    movel([0.147581, -1.249692, -2.655126, -0.807572, 1.570796, 1.718377],accel_mss,speed_ms,0,blend_radius_m)
    movel([0.147363, -1.250802, -2.654535, -0.807052, 1.570796, 1.718159],accel_mss,speed_ms,0,blend_radius_m)
    movel([0.147089, -1.251643, -2.654086, -0.806660, 1.570796, 1.717886],accel_mss,speed_ms,0,blend_radius_m)
    movel([0.145883, -1.253778, -2.652943, -0.805668, 1.570796, 1.716679],accel_mss,speed_ms,0,blend_radius_m)
    movel([0.144114, -1.255772, -2.651871, -0.804746, 1.570796, 1.714911],accel_mss,speed_ms,0,blend_radius_m)
    movel([0.142022, -1.257371, -2.651008, -0.804011, 1.570796, 1.712819],accel_mss,speed_ms,0,blend_radius_m)
    movel([0.139874, -1.258370, -2.650466, -0.803552, 1.570796, 1.710670],accel_mss,speed_ms,0,blend_radius_m)
    movel([0.139347, -1.258581, -2.650352, -0.803456, 1.570796, 1.710143],accel_mss,speed_ms,0,blend_radius_m)
    movel([0.139026, -1.258793, -2.650237, -0.803359, 1.570796, 1.709822],accel_mss,speed_ms,0,blend_radius_m)
    movel([0.138790, -1.259384, -2.649916, -0.803089, 1.570796, 1.709586],accel_mss,speed_ms,0,blend_radius_m)
    movel([0.138626, -1.259915, -2.649627, -0.802847, 1.570796, 1.709423],accel_mss,speed_ms,0,blend_radius_m)
    movel([0.138465, -1.260505, -2.649306, -0.802578, 1.570796, 1.709261],accel_mss,speed_ms,0,blend_radius_m)
    movel([0.138304, -1.261095, -2.648985, -0.802310, 1.570796, 1.709100],accel_mss,speed_ms,0,blend_radius_m)
    movel([0.138138, -1.261625, -2.648695, -0.802069, 1.570796, 1.708934],accel_mss,speed_ms,0,blend_radius_m)
    movel([0.137986, -1.262068, -2.648453, -0.801868, 1.570796, 1.708782],accel_mss,speed_ms,0,blend_radius_m)
    movel([0.137718, -1.262390, -2.648277, -0.801722, 1.570796, 1.708514],accel_mss,speed_ms,0,blend_radius_m)
    movel([0.137358, -1.262485, -2.648225, -0.801679, 1.570796, 1.708154],accel_mss,speed_ms,0,blend_radius_m)
    speed_ms = 0.003
    movel([0.137358, -1.248347, -2.641414, -0.822628, 1.570796, 1.708154],accel_mss,speed_ms,0,blend_radius_m)
    speed_ms = 1.000
    movel([0.137358, -1.221519, -2.627413, -0.863457, 1.570796, 1.708154],accel_mss,speed_ms,0,blend_radius_m)
    movel([0.136331, -1.221369, -2.627491, -0.863529, 1.570796, 1.707127],accel_mss,speed_ms,0,blend_radius_m)
    movel([0.136331, -1.248198, -2.641494, -0.822697, 1.570796, 1.707127],accel_mss,speed_ms,0,blend_radius_m)
    speed_ms = 0.003
    movel([0.136331, -1.258756, -2.646615, -0.807017, 1.570796, 1.707127],accel_mss,speed_ms,0,blend_radius_m)
    speed_ms = 0.007
    movel([0.135965, -1.259022, -2.646471, -0.806896, 1.570796, 1.706761],accel_mss,speed_ms,0,blend_radius_m)
    movel([0.135639, -1.258950, -2.646510, -0.806929, 1.570796, 1.706435],accel_mss,speed_ms,0,blend_radius_m)
    movel([0.135615, -1.258574, -2.646715, -0.807101, 1.570796, 1.706412],accel_mss,speed_ms,0,blend_radius_m)
    movel([0.136097, -1.255221, -2.648532, -0.808636, 1.570796, 1.706894],accel_mss,speed_ms,0,blend_radius_m)
    movel([0.136603, -1.251789, -2.650378, -0.810222, 1.570796, 1.707400],accel_mss,speed_ms,0,blend_radius_m)
    movel([0.136724, -1.251497, -2.650534, -0.810358, 1.570796, 1.707521],accel_mss,speed_ms,0,blend_radius_m)
    movel([0.137247, -1.251196, -2.650695, -0.810498, 1.570796, 1.708044],accel_mss,speed_ms,0,blend_radius_m)
    movel([0.137587, -1.251126, -2.650733, -0.810530, 1.570796, 1.708383],accel_mss,speed_ms,0,blend_radius_m)
    movel([0.137884, -1.251389, -2.650592, -0.810408, 1.570796, 1.708680],accel_mss,speed_ms,0,blend_radius_m)
    movel([0.137821, -1.251968, -2.650282, -0.810139, 1.570796, 1.708618],accel_mss,speed_ms,0,blend_radius_m)
    movel([0.137622, -1.253027, -2.649713, -0.809648, 1.570796, 1.708419],accel_mss,speed_ms,0,blend_radius_m)
    movel([0.137096, -1.255476, -2.648394, -0.808519, 1.570796, 1.707892],accel_mss,speed_ms,0,blend_radius_m)
    movel([0.136830, -1.256677, -2.647744, -0.807968, 1.570796, 1.707626],accel_mss,speed_ms,0,blend_radius_m)
    movel([0.136591, -1.257717, -2.647180, -0.807492, 1.570796, 1.707388],accel_mss,speed_ms,0,blend_radius_m)
    movel([0.136382, -1.258618, -2.646691, -0.807081, 1.570796, 1.707178],accel_mss,speed_ms,0,blend_radius_m)
    speed_ms = 0.003
    movel([0.136331, -1.262337, -2.648306, -0.801746, 1.570796, 1.707127],accel_mss,speed_ms,0,blend_radius_m)
    speed_ms = 0.007
    movel([0.135965, -1.262602, -2.648161, -0.801626, 1.570796, 1.706761],accel_mss,speed_ms,0,blend_radius_m)
    movel([0.135639, -1.262530, -2.648201, -0.801659, 1.570796, 1.706435],accel_mss,speed_ms,0,blend_radius_m)
    movel([0.135615, -1.262155, -2.648406, -0.801828, 1.570796, 1.706412],accel_mss,speed_ms,0,blend_radius_m)
    movel([0.136097, -1.258809, -2.650228, -0.803352, 1.570796, 1.706894],accel_mss,speed_ms,0,blend_radius_m)
    movel([0.136603, -1.255383, -2.652081, -0.804926, 1.570796, 1.707400],accel_mss,speed_ms,0,blend_radius_m)
    movel([0.136724, -1.255092, -2.652237, -0.805060, 1.570796, 1.707521],accel_mss,speed_ms,0,blend_radius_m)
    movel([0.137247, -1.254791, -2.652399, -0.805199, 1.570796, 1.708044],accel_mss,speed_ms,0,blend_radius_m)
    movel([0.137587, -1.254721, -2.652437, -0.805231, 1.570796, 1.708383],accel_mss,speed_ms,0,blend_radius_m)
    movel([0.137884, -1.254983, -2.652296, -0.805110, 1.570796, 1.708680],accel_mss,speed_ms,0,blend_radius_m)
    movel([0.137821, -1.255562, -2.651984, -0.804843, 1.570796, 1.708618],accel_mss,speed_ms,0,blend_radius_m)
    movel([0.137622, -1.256619, -2.651414, -0.804356, 1.570796, 1.708419],accel_mss,speed_ms,0,blend_radius_m)
    movel([0.137096, -1.259063, -2.650090, -0.803235, 1.570796, 1.707892],accel_mss,speed_ms,0,blend_radius_m)
    movel([0.136830, -1.260262, -2.649439, -0.802689, 1.570796, 1.707626],accel_mss,speed_ms,0,blend_radius_m)
    movel([0.136591, -1.261299, -2.648873, -0.802217, 1.570796, 1.707388],accel_mss,speed_ms,0,blend_radius_m)
    movel([0.136382, -1.262199, -2.648382, -0.801809, 1.570796, 1.707178],accel_mss,speed_ms,0,blend_radius_m)
    speed_ms = 0.003
    movel([0.136331, -1.248198, -2.641494, -0.822697, 1.570796, 1.707127],accel_mss,speed_ms,0,blend_radius_m)
    speed_ms = 1.000
    movel([0.136331, -1.221369, -2.627491, -0.863529, 1.570796, 1.707127],accel_mss,speed_ms,0,blend_radius_m)
    movel([0.135518, -1.213284, -2.631635, -0.867470, 1.570796, 1.706315],accel_mss,speed_ms,0,blend_radius_m)
    movel([0.135518, -1.240201, -2.645745, -0.826443, 1.570796, 1.706315],accel_mss,speed_ms,0,blend_radius_m)
    speed_ms = 0.003
    movel([0.135518, -1.250801, -2.650907, -0.810681, 1.570796, 1.706315],accel_mss,speed_ms,0,blend_radius_m)
    speed_ms = 0.007
    movel([0.135184, -1.250928, -2.650838, -0.810622, 1.570796, 1.705981],accel_mss,speed_ms,0,blend_radius_m)
    movel([0.134896, -1.250953, -2.650826, -0.810611, 1.570796, 1.705692],accel_mss,speed_ms,0,blend_radius_m)
    movel([0.134573, -1.250950, -2.650827, -0.810612, 1.570796, 1.705369],accel_mss,speed_ms,0,blend_radius_m)
    movel([0.134262, -1.250915, -2.650845, -0.810628, 1.570796, 1.705059],accel_mss,speed_ms,0,blend_radius_m)
    movel([0.133875, -1.250842, -2.650884, -0.810662, 1.570796, 1.704671],accel_mss,speed_ms,0,blend_radius_m)
    movel([0.133663, -1.250756, -2.650931, -0.810702, 1.570796, 1.704460],accel_mss,speed_ms,0,blend_radius_m)
    movel([0.133527, -1.250440, -2.651099, -0.810849, 1.570796, 1.704323],accel_mss,speed_ms,0,blend_radius_m)
    movel([0.133693, -1.249935, -2.651369, -0.811085, 1.570796, 1.704489],accel_mss,speed_ms,0,blend_radius_m)
    movel([0.134107, -1.249492, -2.651605, -0.811291, 1.570796, 1.704903],accel_mss,speed_ms,0,blend_radius_m)
    movel([0.134658, -1.249246, -2.651736, -0.811407, 1.570796, 1.705455],accel_mss,speed_ms,0,blend_radius_m)
    movel([0.135181, -1.249271, -2.651723, -0.811395, 1.570796, 1.705978],accel_mss,speed_ms,0,blend_radius_m)
    movel([0.135427, -1.249443, -2.651631, -0.811314, 1.570796, 1.706223],accel_mss,speed_ms,0,blend_radius_m)
    movel([0.135661, -1.249807, -2.651437, -0.811145, 1.570796, 1.706457],accel_mss,speed_ms,0,blend_radius_m)
    movel([0.135822, -1.250215, -2.651220, -0.810954, 1.570796, 1.706618],accel_mss,speed_ms,0,blend_radius_m)
    movel([0.135808, -1.250511, -2.651062, -0.810817, 1.570796, 1.706604],accel_mss,speed_ms,0,blend_radius_m)
    movel([0.135518, -1.250801, -2.650907, -0.810681, 1.570796, 1.706315],accel_mss,speed_ms,0,blend_radius_m)
    speed_ms = 0.003
    movel([0.135518, -1.254397, -2.652611, -0.805381, 1.570796, 1.706315],accel_mss,speed_ms,0,blend_radius_m)
    speed_ms = 0.007
    movel([0.135184, -1.254524, -2.652543, -0.805322, 1.570796, 1.705981],accel_mss,speed_ms,0,blend_radius_m)
    movel([0.134896, -1.254548, -2.652530, -0.805311, 1.570796, 1.705692],accel_mss,speed_ms,0,blend_radius_m)
    movel([0.134573, -1.254545, -2.652531, -0.805312, 1.570796, 1.705369],accel_mss,speed_ms,0,blend_radius_m)
    movel([0.134262, -1.254511, -2.652550, -0.805328, 1.570796, 1.705059],accel_mss,speed_ms,0,blend_radius_m)
    movel([0.133875, -1.254438, -2.652589, -0.805362, 1.570796, 1.704671],accel_mss,speed_ms,0,blend_radius_m)
    movel([0.133663, -1.254352, -2.652635, -0.805402, 1.570796, 1.704460],accel_mss,speed_ms,0,blend_radius_m)
    movel([0.133527, -1.254037, -2.652804, -0.805548, 1.570796, 1.704323],accel_mss,speed_ms,0,blend_radius_m)
    movel([0.133693, -1.253533, -2.653075, -0.805781, 1.570796, 1.704489],accel_mss,speed_ms,0,blend_radius_m)
    movel([0.134107, -1.253091, -2.653312, -0.805987, 1.570796, 1.704903],accel_mss,speed_ms,0,blend_radius_m)
    movel([0.134658, -1.252845, -2.653444, -0.806101, 1.570796, 1.705455],accel_mss,speed_ms,0,blend_radius_m)
    movel([0.135181, -1.252869, -2.653430, -0.806089, 1.570796, 1.705978],accel_mss,speed_ms,0,blend_radius_m)
    movel([0.135427, -1.253041, -2.653338, -0.806009, 1.570796, 1.706223],accel_mss,speed_ms,0,blend_radius_m)
    movel([0.135661, -1.253405, -2.653143, -0.805841, 1.570796, 1.706457],accel_mss,speed_ms,0,blend_radius_m)
    movel([0.135822, -1.253812, -2.652925, -0.805652, 1.570796, 1.706618],accel_mss,speed_ms,0,blend_radius_m)
    movel([0.135808, -1.254107, -2.652767, -0.805515, 1.570796, 1.706604],accel_mss,speed_ms,0,blend_radius_m)
    movel([0.135518, -1.254397, -2.652611, -0.805381, 1.570796, 1.706315],accel_mss,speed_ms,0,blend_radius_m)
    speed_ms = 0.003
    movel([0.135518, -1.240201, -2.645745, -0.826443, 1.570796, 1.706315],accel_mss,speed_ms,0,blend_radius_m)
    speed_ms = 1.000
    movel([0.135518, -1.213284, -2.631635, -0.867470, 1.570796, 1.706315],accel_mss,speed_ms,0,blend_radius_m)
    movel([0.139093, -1.211934, -2.632319, -0.868135, 1.570796, 1.709889],accel_mss,speed_ms,0,blend_radius_m)
    movel([0.139093, -1.238865, -2.646447, -0.827076, 1.570796, 1.709889],accel_mss,speed_ms,0,blend_radius_m)
    speed_ms = 0.003
    movel([0.139093, -1.249472, -2.651616, -0.811301, 1.570796, 1.709889],accel_mss,speed_ms,0,blend_radius_m)
    speed_ms = 0.007
    movel([0.139118, -1.249017, -2.651858, -0.811513, 1.570796, 1.709914],accel_mss,speed_ms,0,blend_radius_m)
    movel([0.139248, -1.248505, -2.652131, -0.811753, 1.570796, 1.710045],accel_mss,speed_ms,0,blend_radius_m)
    movel([0.139468, -1.248099, -2.652347, -0.811943, 1.570796, 1.710264],accel_mss,speed_ms,0,blend_radius_m)
    movel([0.139744, -1.247818, -2.652496, -0.812075, 1.570796, 1.710540],accel_mss,speed_ms,0,blend_radius_m)
    movel([0.140071, -1.247632, -2.652595, -0.812162, 1.570796, 1.710868],accel_mss,speed_ms,0,blend_radius_m)
    movel([0.140367, -1.247587, -2.652619, -0.812183, 1.570796, 1.711163],accel_mss,speed_ms,0,blend_radius_m)
    movel([0.140630, -1.247982, -2.652409, -0.811998, 1.570796, 1.711426],accel_mss,speed_ms,0,blend_radius_m)
    movel([0.140571, -1.248308, -2.652236, -0.811845, 1.570796, 1.711368],accel_mss,speed_ms,0,blend_radius_m)
    movel([0.140360, -1.248691, -2.652032, -0.811666, 1.570796, 1.711157],accel_mss,speed_ms,0,blend_radius_m)
    movel([0.139989, -1.249142, -2.651792, -0.811455, 1.570796, 1.710786],accel_mss,speed_ms,0,blend_radius_m)
    movel([0.139673, -1.249473, -2.651615, -0.811300, 1.570796, 1.710469],accel_mss,speed_ms,0,blend_radius_m)
    movel([0.139344, -1.249692, -2.651499, -0.811198, 1.570796, 1.710140],accel_mss,speed_ms,0,blend_radius_m)
    movel([0.139093, -1.249472, -2.651616, -0.811301, 1.570796, 1.709889],accel_mss,speed_ms,0,blend_radius_m)
    speed_ms = 0.003
    movel([0.139093, -1.253071, -2.653322, -0.805996, 1.570796, 1.709889],accel_mss,speed_ms,0,blend_radius_m)
    speed_ms = 0.007
    movel([0.139118, -1.252616, -2.653566, -0.806207, 1.570796, 1.709914],accel_mss,speed_ms,0,blend_radius_m)
    movel([0.139248, -1.252105, -2.653839, -0.806445, 1.570796, 1.710045],accel_mss,speed_ms,0,blend_radius_m)
    movel([0.139468, -1.251700, -2.654056, -0.806633, 1.570796, 1.710264],accel_mss,speed_ms,0,blend_radius_m)
    movel([0.139744, -1.251419, -2.654206, -0.806764, 1.570796, 1.710540],accel_mss,speed_ms,0,blend_radius_m)
    movel([0.140071, -1.251234, -2.654304, -0.806851, 1.570796, 1.710868],accel_mss,speed_ms,0,blend_radius_m)
    movel([0.140367, -1.251188, -2.654329, -0.806872, 1.570796, 1.711163],accel_mss,speed_ms,0,blend_radius_m)
    movel([0.140630, -1.251583, -2.654118, -0.806688, 1.570796, 1.711426],accel_mss,speed_ms,0,blend_radius_m)
    movel([0.140571, -1.251909, -2.653944, -0.806536, 1.570796, 1.711368],accel_mss,speed_ms,0,blend_radius_m)
    movel([0.140360, -1.252291, -2.653740, -0.806358, 1.570796, 1.711157],accel_mss,speed_ms,0,blend_radius_m)
    movel([0.139989, -1.252740, -2.653499, -0.806149, 1.570796, 1.710786],accel_mss,speed_ms,0,blend_radius_m)
    movel([0.139673, -1.253072, -2.653322, -0.805995, 1.570796, 1.710469],accel_mss,speed_ms,0,blend_radius_m)
    movel([0.139344, -1.253290, -2.653205, -0.805894, 1.570796, 1.710140],accel_mss,speed_ms,0,blend_radius_m)
    movel([0.139093, -1.253071, -2.653322, -0.805996, 1.570796, 1.709889],accel_mss,speed_ms,0,blend_radius_m)
    speed_ms = 0.003
    movel([0.139093, -1.238865, -2.646447, -0.827076, 1.570796, 1.709889],accel_mss,speed_ms,0,blend_radius_m)
    speed_ms = 1.000
    movel([0.139093, -1.211934, -2.632319, -0.868135, 1.570796, 1.709889],accel_mss,speed_ms,0,blend_radius_m)
    movel([0.082807, -1.213918, -2.631313, -0.867159, 1.570796, 1.653603],accel_mss,speed_ms,0,blend_radius_m)
    movel([0.082807, -1.240828, -2.645414, -0.826147, 1.570796, 1.653603],accel_mss,speed_ms,0,blend_radius_m)
    speed_ms = 0.003
    movel([0.082807, -1.251425, -2.650573, -0.810391, 1.570796, 1.653603],accel_mss,speed_ms,0,blend_radius_m)
    speed_ms = 0.007
    movel([0.081255, -1.253623, -2.649393, -0.809373, 1.570796, 1.652051],accel_mss,speed_ms,0,blend_radius_m)
    movel([0.079525, -1.256064, -2.648076, -0.808249, 1.570796, 1.650321],accel_mss,speed_ms,0,blend_radius_m)
    movel([0.077484, -1.258933, -2.646519, -0.806937, 1.570796, 1.648280],accel_mss,speed_ms,0,blend_radius_m)
    movel([0.074500, -1.263106, -2.644237, -0.805046, 1.570796, 1.645296],accel_mss,speed_ms,0,blend_radius_m)
    movel([0.072945, -1.265220, -2.643072, -0.804097, 1.570796, 1.643742],accel_mss,speed_ms,0,blend_radius_m)
    movel([0.072027, -1.266399, -2.642421, -0.803570, 1.570796, 1.642823],accel_mss,speed_ms,0,blend_radius_m)
    movel([0.072454, -1.264954, -2.643219, -0.804216, 1.570796, 1.643251],accel_mss,speed_ms,0,blend_radius_m)
    movel([0.073107, -1.263398, -2.644076, -0.804915, 1.570796, 1.643903],accel_mss,speed_ms,0,blend_radius_m)
    movel([0.073883, -1.261564, -2.645082, -0.805742, 1.570796, 1.644679],accel_mss,speed_ms,0,blend_radius_m)
    movel([0.074867, -1.259224, -2.646361, -0.806804, 1.570796, 1.645663],accel_mss,speed_ms,0,blend_radius_m)
    movel([0.075443, -1.257792, -2.647140, -0.807458, 1.570796, 1.646239],accel_mss,speed_ms,0,blend_radius_m)
    movel([0.075810, -1.256811, -2.647672, -0.807906, 1.570796, 1.646606],accel_mss,speed_ms,0,blend_radius_m)
    movel([0.075634, -1.256569, -2.647803, -0.808017, 1.570796, 1.646430],accel_mss,speed_ms,0,blend_radius_m)
    movel([0.075253, -1.256647, -2.647761, -0.807982, 1.570796, 1.646050],accel_mss,speed_ms,0,blend_radius_m)
    movel([0.074598, -1.256851, -2.647650, -0.807888, 1.570796, 1.645394],accel_mss,speed_ms,0,blend_radius_m)
    movel([0.073341, -1.257289, -2.647413, -0.807688, 1.570796, 1.644137],accel_mss,speed_ms,0,blend_radius_m)
    movel([0.072270, -1.257663, -2.647210, -0.807516, 1.570796, 1.643066],accel_mss,speed_ms,0,blend_radius_m)
    movel([0.071543, -1.257893, -2.647085, -0.807411, 1.570796, 1.642339],accel_mss,speed_ms,0,blend_radius_m)
    movel([0.071034, -1.258033, -2.647009, -0.807347, 1.570796, 1.641830],accel_mss,speed_ms,0,blend_radius_m)
    movel([0.070865, -1.257859, -2.647103, -0.807427, 1.570796, 1.641661],accel_mss,speed_ms,0,blend_radius_m)
    movel([0.071306, -1.256707, -2.647728, -0.807954, 1.570796, 1.642103],accel_mss,speed_ms,0,blend_radius_m)
    movel([0.071948, -1.255121, -2.648586, -0.808682, 1.570796, 1.642744],accel_mss,speed_ms,0,blend_radius_m)
    movel([0.072961, -1.252711, -2.649883, -0.809795, 1.570796, 1.643757],accel_mss,speed_ms,0,blend_radius_m)
    movel([0.073821, -1.250693, -2.650965, -0.810732, 1.570796, 1.644617],accel_mss,speed_ms,0,blend_radius_m)
    movel([0.074573, -1.248951, -2.651893, -0.811544, 1.570796, 1.645369],accel_mss,speed_ms,0,blend_radius_m)
    movel([0.075236, -1.247422, -2.652706, -0.812261, 1.570796, 1.646032],accel_mss,speed_ms,0,blend_radius_m)
    movel([0.075486, -1.247116, -2.652869, -0.812405, 1.570796, 1.646282],accel_mss,speed_ms,0,blend_radius_m)
    movel([0.076173, -1.246818, -2.653027, -0.812545, 1.570796, 1.646970],accel_mss,speed_ms,0,blend_radius_m)
    movel([0.077201, -1.246406, -2.653245, -0.812738, 1.570796, 1.647997],accel_mss,speed_ms,0,blend_radius_m)
    movel([0.078902, -1.245763, -2.653585, -0.813041, 1.570796, 1.649699],accel_mss,speed_ms,0,blend_radius_m)
    movel([0.080795, -1.245067, -2.653953, -0.813370, 1.570796, 1.651591],accel_mss,speed_ms,0,blend_radius_m)
    movel([0.081727, -1.244749, -2.654120, -0.813520, 1.570796, 1.652524],accel_mss,speed_ms,0,blend_radius_m)
    movel([0.082276, -1.244594, -2.654202, -0.813593, 1.570796, 1.653072],accel_mss,speed_ms,0,blend_radius_m)
    movel([0.082396, -1.244795, -2.654096, -0.813498, 1.570796, 1.653193],accel_mss,speed_ms,0,blend_radius_m)
    movel([0.081838, -1.245860, -2.653533, -0.812995, 1.570796, 1.652635],accel_mss,speed_ms,0,blend_radius_m)
    movel([0.081159, -1.247118, -2.652868, -0.812404, 1.570796, 1.651955],accel_mss,speed_ms,0,blend_radius_m)
    movel([0.080328, -1.248601, -2.652080, -0.811708, 1.570796, 1.651124],accel_mss,speed_ms,0,blend_radius_m)
    movel([0.079241, -1.250532, -2.651050, -0.810807, 1.570796, 1.650037],accel_mss,speed_ms,0,blend_radius_m)
    movel([0.078655, -1.251629, -2.650463, -0.810296, 1.570796, 1.649451],accel_mss,speed_ms,0,blend_radius_m)
    movel([0.078314, -1.252329, -2.650088, -0.809972, 1.570796, 1.649110],accel_mss,speed_ms,0,blend_radius_m)
    movel([0.078472, -1.252579, -2.649954, -0.809856, 1.570796, 1.649269],accel_mss,speed_ms,0,blend_radius_m)
    movel([0.078805, -1.252519, -2.649986, -0.809884, 1.570796, 1.649601],accel_mss,speed_ms,0,blend_radius_m)
    movel([0.079378, -1.252348, -2.650078, -0.809963, 1.570796, 1.650175],accel_mss,speed_ms,0,blend_radius_m)
    movel([0.080470, -1.251972, -2.650280, -0.810137, 1.570796, 1.651266],accel_mss,speed_ms,0,blend_radius_m)
    movel([0.081795, -1.251513, -2.650525, -0.810350, 1.570796, 1.652591],accel_mss,speed_ms,0,blend_radius_m)
    movel([0.082424, -1.251323, -2.650627, -0.810439, 1.570796, 1.653221],accel_mss,speed_ms,0,blend_radius_m)
    movel([0.082757, -1.251264, -2.650659, -0.810466, 1.570796, 1.653553],accel_mss,speed_ms,0,blend_radius_m)
    speed_ms = 0.003
    movel([0.082807, -1.255019, -2.652276, -0.805093, 1.570796, 1.653603],accel_mss,speed_ms,0,blend_radius_m)
    speed_ms = 0.007
    movel([0.081255, -1.257214, -2.651093, -0.804083, 1.570796, 1.652051],accel_mss,speed_ms,0,blend_radius_m)
    movel([0.079525, -1.259650, -2.649772, -0.802968, 1.570796, 1.650321],accel_mss,speed_ms,0,blend_radius_m)
    movel([0.077484, -1.262513, -2.648210, -0.801666, 1.570796, 1.648280],accel_mss,speed_ms,0,blend_radius_m)
    movel([0.074500, -1.266678, -2.645920, -0.799791, 1.570796, 1.645296],accel_mss,speed_ms,0,blend_radius_m)
    movel([0.072945, -1.268788, -2.644752, -0.798849, 1.570796, 1.643742],accel_mss,speed_ms,0,blend_radius_m)
    movel([0.072027, -1.269965, -2.644098, -0.798326, 1.570796, 1.642823],accel_mss,speed_ms,0,blend_radius_m)
    movel([0.072454, -1.268522, -2.644899, -0.798967, 1.570796, 1.643251],accel_mss,speed_ms,0,blend_radius_m)
    movel([0.073107, -1.266970, -2.645759, -0.799660, 1.570796, 1.643903],accel_mss,speed_ms,0,blend_radius_m)
    movel([0.073883, -1.265139, -2.646768, -0.800481, 1.570796, 1.644679],accel_mss,speed_ms,0,blend_radius_m)
    movel([0.074867, -1.262803, -2.648051, -0.801535, 1.570796, 1.645663],accel_mss,speed_ms,0,blend_radius_m)
    movel([0.075443, -1.261374, -2.648832, -0.802183, 1.570796, 1.646239],accel_mss,speed_ms,0,blend_radius_m)
    movel([0.075810, -1.260395, -2.649366, -0.802628, 1.570796, 1.646606],accel_mss,speed_ms,0,blend_radius_m)
    movel([0.075634, -1.260153, -2.649498, -0.802738, 1.570796, 1.646430],accel_mss,speed_ms,0,blend_radius_m)
    movel([0.075253, -1.260231, -2.649455, -0.802702, 1.570796, 1.646050],accel_mss,speed_ms,0,blend_radius_m)
    movel([0.074598, -1.260436, -2.649344, -0.802609, 1.570796, 1.645394],accel_mss,speed_ms,0,blend_radius_m)
    movel([0.073341, -1.260872, -2.649106, -0.802411, 1.570796, 1.644137],accel_mss,speed_ms,0,blend_radius_m)
    movel([0.072270, -1.261246, -2.648902, -0.802241, 1.570796, 1.643066],accel_mss,speed_ms,0,blend_radius_m)
    movel([0.071543, -1.261476, -2.648777, -0.802136, 1.570796, 1.642339],accel_mss,speed_ms,0,blend_radius_m)
    movel([0.071034, -1.261615, -2.648701, -0.802073, 1.570796, 1.641830],accel_mss,speed_ms,0,blend_radius_m)
    movel([0.070865, -1.261441, -2.648796, -0.802152, 1.570796, 1.641661],accel_mss,speed_ms,0,blend_radius_m)
    movel([0.071306, -1.260292, -2.649422, -0.802675, 1.570796, 1.642103],accel_mss,speed_ms,0,blend_radius_m)
    movel([0.071948, -1.258709, -2.650283, -0.803397, 1.570796, 1.642744],accel_mss,speed_ms,0,blend_radius_m)
    movel([0.072961, -1.256303, -2.651584, -0.804501, 1.570796, 1.643757],accel_mss,speed_ms,0,blend_radius_m)
    movel([0.073821, -1.254289, -2.652669, -0.805431, 1.570796, 1.644617],accel_mss,speed_ms,0,blend_radius_m)
    movel([0.074573, -1.252551, -2.653601, -0.806237, 1.570796, 1.645369],accel_mss,speed_ms,0,blend_radius_m)
    movel([0.075236, -1.251024, -2.654416, -0.806948, 1.570796, 1.646032],accel_mss,speed_ms,0,blend_radius_m)
    movel([0.075486, -1.250718, -2.654579, -0.807091, 1.570796, 1.646282],accel_mss,speed_ms,0,blend_radius_m)
    movel([0.076173, -1.250421, -2.654738, -0.807230, 1.570796, 1.646970],accel_mss,speed_ms,0,blend_radius_m)
    movel([0.077201, -1.250010, -2.654957, -0.807423, 1.570796, 1.647997],accel_mss,speed_ms,0,blend_radius_m)
    movel([0.078902, -1.249368, -2.655298, -0.807723, 1.570796, 1.649699],accel_mss,speed_ms,0,blend_radius_m)
    movel([0.080795, -1.248673, -2.655667, -0.808049, 1.570796, 1.651591],accel_mss,speed_ms,0,blend_radius_m)
    movel([0.081727, -1.248356, -2.655835, -0.808198, 1.570796, 1.652524],accel_mss,speed_ms,0,blend_radius_m)
    movel([0.082276, -1.248201, -2.655917, -0.808271, 1.570796, 1.653072],accel_mss,speed_ms,0,blend_radius_m)
    movel([0.082396, -1.248402, -2.655810, -0.808176, 1.570796, 1.653193],accel_mss,speed_ms,0,blend_radius_m)
    movel([0.081838, -1.249465, -2.655246, -0.807678, 1.570796, 1.652635],accel_mss,speed_ms,0,blend_radius_m)
    movel([0.081159, -1.250720, -2.654578, -0.807090, 1.570796, 1.651955],accel_mss,speed_ms,0,blend_radius_m)
    movel([0.080328, -1.252201, -2.653788, -0.806400, 1.570796, 1.651124],accel_mss,speed_ms,0,blend_radius_m)
    movel([0.079241, -1.254128, -2.652755, -0.805506, 1.570796, 1.650037],accel_mss,speed_ms,0,blend_radius_m)
    movel([0.078655, -1.255224, -2.652166, -0.804999, 1.570796, 1.649451],accel_mss,speed_ms,0,blend_radius_m)
    movel([0.078314, -1.255922, -2.651790, -0.804677, 1.570796, 1.649110],accel_mss,speed_ms,0,blend_radius_m)
    movel([0.078472, -1.256172, -2.651655, -0.804562, 1.570796, 1.649269],accel_mss,speed_ms,0,blend_radius_m)
    movel([0.078805, -1.256112, -2.651688, -0.804589, 1.570796, 1.649601],accel_mss,speed_ms,0,blend_radius_m)
    movel([0.079378, -1.255941, -2.651780, -0.804668, 1.570796, 1.650175],accel_mss,speed_ms,0,blend_radius_m)
    movel([0.080470, -1.255566, -2.651982, -0.804841, 1.570796, 1.651266],accel_mss,speed_ms,0,blend_radius_m)
    movel([0.081795, -1.255108, -2.652228, -0.805053, 1.570796, 1.652591],accel_mss,speed_ms,0,blend_radius_m)
    movel([0.082424, -1.254918, -2.652331, -0.805140, 1.570796, 1.653221],accel_mss,speed_ms,0,blend_radius_m)
    movel([0.082757, -1.254859, -2.652362, -0.805167, 1.570796, 1.653553],accel_mss,speed_ms,0,blend_radius_m)
    speed_ms = 0.003
    movel([0.082807, -1.240828, -2.645414, -0.826147, 1.570796, 1.653603],accel_mss,speed_ms,0,blend_radius_m)
    speed_ms = 1.000
    movel([0.082807, -1.213918, -2.631313, -0.867159, 1.570796, 1.653603],accel_mss,speed_ms,0,blend_radius_m)
    movel([0.061043, -1.170670, -2.652297, -0.889422, 1.570796, 1.631840],accel_mss,speed_ms,0,blend_radius_m)
    movel([0.061043, -1.077942, -2.586592, -1.047856, 1.570796, 1.631840],accel_mss,speed_ms,0,blend_radius_m)
    # End of main program
  end

  Machining1()
end
